FUNCTION_BLOCK Metadata IMPLEMENTS I_Metadata
VAR
	metadata : Stack;
END_VAR

METHOD PUBLIC GetEnumerator : I_ForwardEnumerator
VAR_INPUT
END_VAR
GetEnumerator := metadata.GetEnumerator();
END_METHOD

METHOD PUBLIC Insert
VAR_INPUT
	MetadatumToAdd : I_Metadatum;
END_VAR
metadata.Push(MetadatumToAdd);
END_METHOD

METHOD PUBLIC TryGetByName : BOOL
VAR_INPUT
	Name : STRING;
	Destination : REFERENCE TO I_Metadatum;
END_VAR
VAR
	metadatumEnumerator : I_ForwardEnumerator;
	currentMetadatum : I_Metadatum;
END_VAR
metadatumEnumerator := metadata.GetEnumerator();

WHILE metadatumEnumerator.MoveNext() DO 
	IF NOT metadatumEnumerator.TryGet(currentMetadatum) THEN
		CONTINUE;
	END_IF
	
	IF currentMetadatum.Name = Name THEN 
		TryGetByName := TRUE;
		Destination := currentMetadatum;
		EXIT;
	END_IF

END_WHILE

metadatumEnumerator.Dispose();
END_METHOD

END_FUNCTION_BLOCK

(* stored: Version 1.1.0.1, ProductVersion 3.1.4024.12
   POU Metadata: Id {d4b0ff48-d878-04ac-1814-bf7a496cd6c1}, SpecialFunc None
   Method GetEnumerator: Id {b3e14664-f931-0abc-3a9e-83b712e76bcc}
   Method Insert: Id {912794a7-c6b6-050e-2b3f-1470aef8d028}
   Method TryGetByName: Id {cbaf7bca-e459-0b60-310e-3808dd545bde} *)
